PROGRAM MAIN
VAR

END_VAR

END_PROGRAM

(* stored: Version 1.1.0.1, ProductVersion 3.1.4024.15
   POU MAIN: Id {cce30028-973b-43e0-9926-98c587a2f51b}, SpecialFunc None *)
